PROGRAM PRG_SFLX_ValidationAsConfirmation
VAR
	rtrigValidCameraTrigger				: F_TRIG;
	bSideFlexValidCameraTrigger			: BOOL;

	rsSideFlexTwoOutersInAggregation	: RS;
	rsSideFlexPackToOuterProcessing		: RS;

	rtrigNewOuterArrived					: R_TRIG;
	bNewOuterIsProccesing				: BOOL;
	tonValidationTimout					: TON;
	bValidationTimeout					: BOOL;
	bValidationTimeoutReset				: BOOL;
	fbTimeoutCounter						: CTU;
	nCount									: WORD;


	fbOuterValidationCamera				: FB_SCANNER_CameraSelect;
	(*stOuterValidationCameraOptions		: ST_SCANNER_Options := (eScannerType := E_MV_420_FULL, nImageBuffer := 1, nExpectedResp := 2);*)
	fbOuterValidationEvaluation		: FB_SCANNER_Evaluation;

	fbCheckForDuplicateOuterValidation	: FB_OUTER_CheckDuplicateStatus;


	rtrigOuterValidationCameraDone				: R_TRIG;
	bOuterValidationCameraDone				: BOOL;
	bDataReadyForValidation			: BOOL;
	bQAReject							: BOOL;

	sLastImageLableString				: T_OUTER_Barcode;

	fbPerformance							: FB_Interval;
	fbMoveOuterData						: FB_OUTER_MoveOuterStatus;
	fbCompleteOuterFromQueue			: FB_OUTER_CompleteDataFromQueue_NoCam;
	fbMETSValidateOuterForReject			: FB_OUTER_ValidateOuterForReject;
	tofValidateOuterDoneForHMI			: TOF;
	fbMasterListUpdate					: FB_OUTER_MasterListUpdate;

	stLastOuterCompleted				: ST_OUTER_Status;
	sLastReadOuterBarcode			: T_OUTER_Barcode;
	nOutersCompleted					: UDINT;
	bDoneInfo							: BOOL;

	rtrigSetOuterValidationOK			: R_TRIG;
	rtrigSetOuterValidationNOK		: R_TRIG;

	rsOuterRejectStation 				: RS;
	rsOuterRejectConfirmation 		: RS;

	rtrigResetValidationStatus			: R_TRIG;

	sRejectCode						: STRING(255);
	fbArchiveInvalidOuters			: FB_OUTER_ArchiveInvalidOuters;
	aReasonForReject					: ARRAY[0..50] OF STRING(255);
	bClearList							: BOOL;

	fbOuterProduced					: FB_KPI_GenericEfficiency;
	fbOuterInspection					: FB_KPI_OutersEfficiency;

	stDummyImage					: ST_SCANNER_ImageData;

	fbOuterLevelCounter				: FB_KPI_OuterLevelCounter;

	fbQARejectCounter				: FB_CTU32;
	fbOuterValidationIndexOK			: FB_CTU32;

	ctuConsecutiveOuterRejects		: CTU;
	nActualCount						: WORD;
END_VAR
VAR // added by the converter: edge detectors and wires of the graphical bodies
    _w1 : E_CYLINDER_Position;
    _w2, _w3 : BOOL;
END_VAR

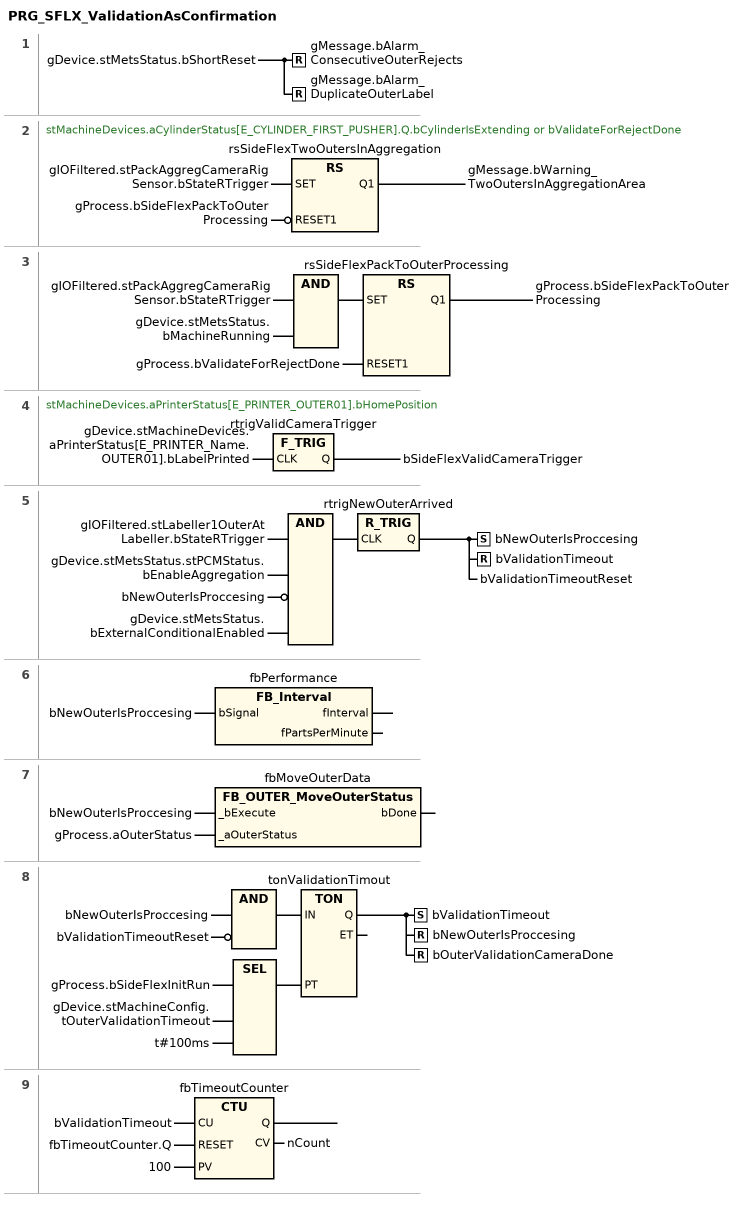
// NETWORK 1
gMessage.bAlarm_ConsecutiveOuterRejects R= gDevice.stMetsStatus.bShortReset;
gMessage.bAlarm_DuplicateOuterLabel R= gDevice.stMetsStatus.bShortReset;

// NETWORK 2
// stMachineDevices.aCylinderStatus[E_CYLINDER_FIRST_PUSHER].Q.bCylinderIsExtending or bValidateForRejectDone
rsSideFlexTwoOutersInAggregation(SET := gIOFiltered.stPackAggregCameraRigSensor.bStateRTrigger, RESET1 := NOT gProcess.bSideFlexPackToOuterProcessing); // RS
gMessage.bWarning_TwoOutersInAggregationArea := rsSideFlexTwoOutersInAggregation.Q1;

// NETWORK 3
rsSideFlexPackToOuterProcessing(SET := gIOFiltered.stPackAggregCameraRigSensor.bStateRTrigger AND gDevice.stMetsStatus.bMachineRunning, RESET1 := gProcess.bValidateForRejectDone); // RS
gProcess.bSideFlexPackToOuterProcessing := rsSideFlexPackToOuterProcessing.Q1;

// NETWORK 4
// stMachineDevices.aPrinterStatus[E_PRINTER_OUTER01].bHomePosition
rtrigValidCameraTrigger(CLK := gDevice.stMachineDevices.aPrinterStatus[E_PRINTER_Name.OUTER01].bLabelPrinted); // F_TRIG
bSideFlexValidCameraTrigger := rtrigValidCameraTrigger.Q;

// NETWORK 5
rtrigNewOuterArrived(CLK := gIOFiltered.stLabeller1OuterAtLabeller.bStateRTrigger AND gDevice.stMetsStatus.stPCMStatus.bEnableAggregation AND NOT bNewOuterIsProccesing AND gDevice.stMetsStatus.bExternalConditionalEnabled); // R_TRIG
bNewOuterIsProccesing S= rtrigNewOuterArrived.Q;
bValidationTimeout R= rtrigNewOuterArrived.Q;
bValidationTimeoutReset := rtrigNewOuterArrived.Q;

// NETWORK 6
fbPerformance(bSignal := bNewOuterIsProccesing); // FB_Interval

// NETWORK 7
fbMoveOuterData(_bExecute := bNewOuterIsProccesing, _aOuterStatus := gProcess.aOuterStatus); // FB_OUTER_MoveOuterStatus

// NETWORK 8
tonValidationTimout(IN := bNewOuterIsProccesing AND NOT bValidationTimeoutReset, PT := SEL(gProcess.bSideFlexInitRun, gDevice.stMachineConfig.tOuterValidationTimeout, t#100ms)); // TON
bValidationTimeout S= tonValidationTimout.Q;
bNewOuterIsProccesing R= tonValidationTimout.Q;
bOuterValidationCameraDone R= tonValidationTimout.Q;

// NETWORK 9
fbTimeoutCounter(CU := bValidationTimeout, RESET := fbTimeoutCounter.Q, PV := 100, CV => nCount); // CTU

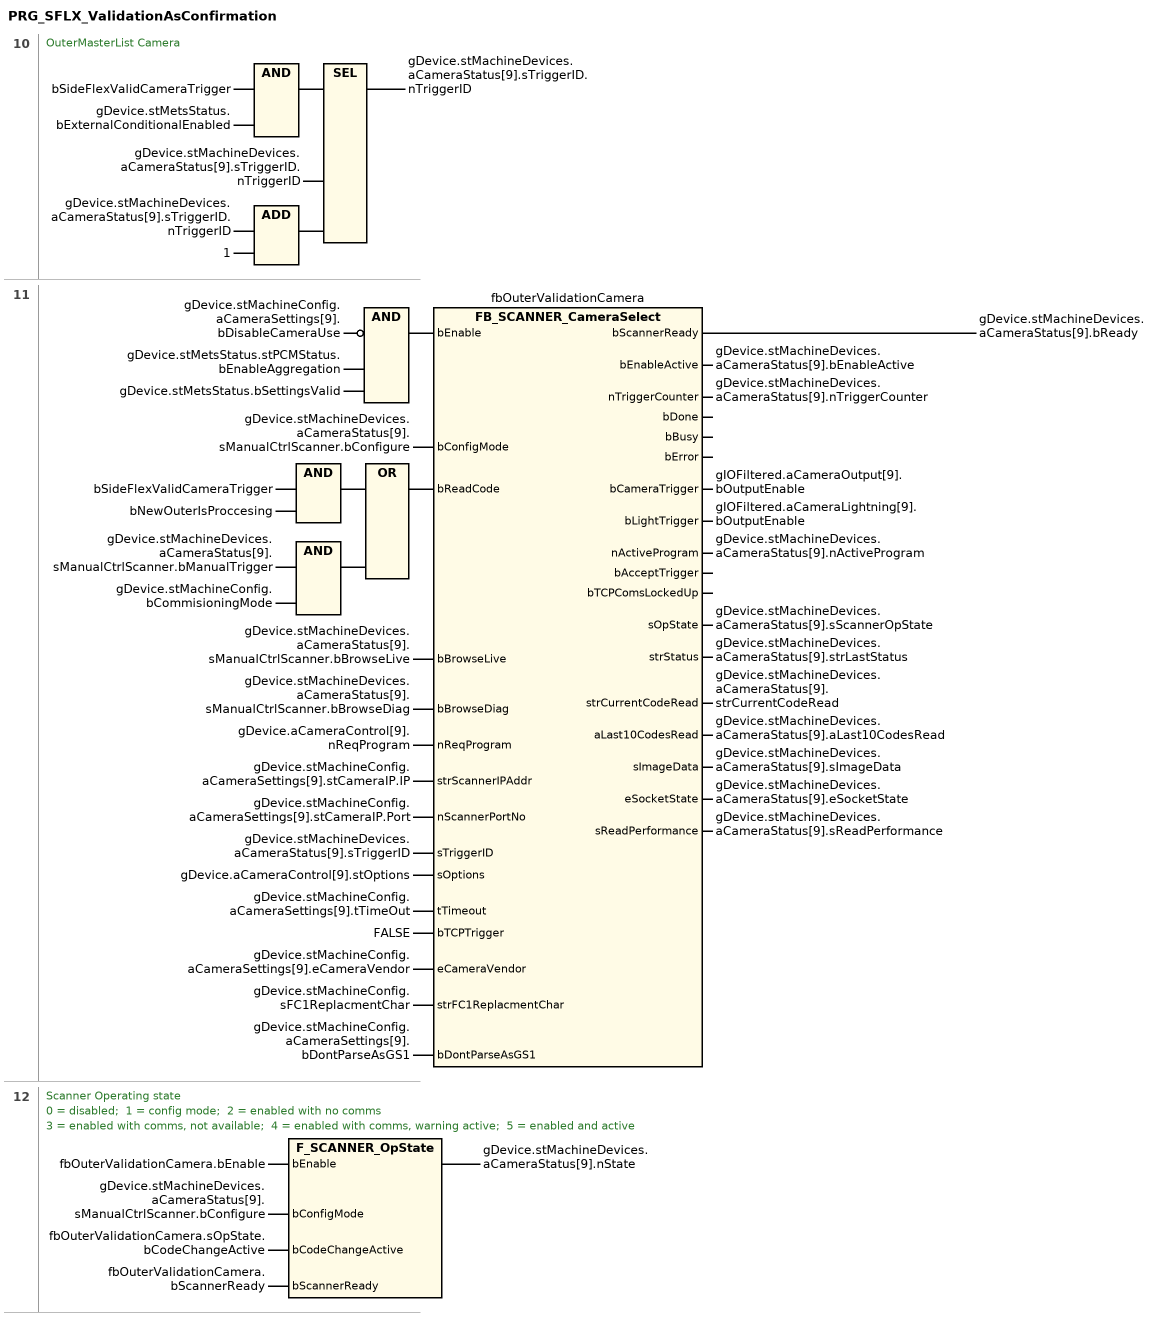
// NETWORK 10
// OuterMasterList Camera
gDevice.stMachineDevices.aCameraStatus[9].sTriggerID.nTriggerID := SEL(bSideFlexValidCameraTrigger AND gDevice.stMetsStatus.bExternalConditionalEnabled, gDevice.stMachineDevices.aCameraStatus[9].sTriggerID.nTriggerID, gDevice.stMachineDevices.aCameraStatus[9].sTriggerID.nTriggerID + 1);

// NETWORK 11
fbOuterValidationCamera(
    bEnable := NOT gDevice.stMachineConfig.aCameraSettings[9].bDisableCameraUse AND gDevice.stMetsStatus.stPCMStatus.bEnableAggregation AND gDevice.stMetsStatus.bSettingsValid,
    bConfigMode := gDevice.stMachineDevices.aCameraStatus[9].sManualCtrlScanner.bConfigure,
    bReadCode := bSideFlexValidCameraTrigger AND bNewOuterIsProccesing OR gDevice.stMachineDevices.aCameraStatus[9].sManualCtrlScanner.bManualTrigger AND gDevice.stMachineConfig.bCommisioningMode,
    bBrowseLive := gDevice.stMachineDevices.aCameraStatus[9].sManualCtrlScanner.bBrowseLive,
    bBrowseDiag := gDevice.stMachineDevices.aCameraStatus[9].sManualCtrlScanner.bBrowseDiag,
    nReqProgram := gDevice.aCameraControl[9].nReqProgram,
    strScannerIPAddr := gDevice.stMachineConfig.aCameraSettings[9].stCameraIP.IP,
    nScannerPortNo := gDevice.stMachineConfig.aCameraSettings[9].stCameraIP.Port,
    sTriggerID := gDevice.stMachineDevices.aCameraStatus[9].sTriggerID,
    sOptions := gDevice.aCameraControl[9].stOptions,
    tTimeout := gDevice.stMachineConfig.aCameraSettings[9].tTimeOut,
    bTCPTrigger := FALSE,
    eCameraVendor := gDevice.stMachineConfig.aCameraSettings[9].eCameraVendor,
    strFC1ReplacmentChar := gDevice.stMachineConfig.sFC1ReplacmentChar,
    bDontParseAsGS1 := gDevice.stMachineConfig.aCameraSettings[9].bDontParseAsGS1,
    bEnableActive => gDevice.stMachineDevices.aCameraStatus[9].bEnableActive,
    nTriggerCounter => gDevice.stMachineDevices.aCameraStatus[9].nTriggerCounter,
    bCameraTrigger => gIOFiltered.aCameraOutput[9].bOutputEnable,
    bLightTrigger => gIOFiltered.aCameraLightning[9].bOutputEnable,
    nActiveProgram => gDevice.stMachineDevices.aCameraStatus[9].nActiveProgram,
    sOpState => gDevice.stMachineDevices.aCameraStatus[9].sScannerOpState,
    strStatus => gDevice.stMachineDevices.aCameraStatus[9].strLastStatus,
    strCurrentCodeRead => gDevice.stMachineDevices.aCameraStatus[9].strCurrentCodeRead,
    aLast10CodesRead => gDevice.stMachineDevices.aCameraStatus[9].aLast10CodesRead,
    sImageData => gDevice.stMachineDevices.aCameraStatus[9].sImageData,
    eSocketState => gDevice.stMachineDevices.aCameraStatus[9].eSocketState,
    sReadPerformance => gDevice.stMachineDevices.aCameraStatus[9].sReadPerformance); // FB_SCANNER_CameraSelect
gDevice.stMachineDevices.aCameraStatus[9].bReady := fbOuterValidationCamera.bScannerReady;

// NETWORK 12
// 					Scanner Operating state
// 0 = disabled;  1 = config mode;  2 = enabled with no comms
// 3 = enabled with comms, not available;  4 = enabled with comms, warning active;  5 = enabled and active
//
gDevice.stMachineDevices.aCameraStatus[9].nState := F_SCANNER_OpState(bEnable := fbOuterValidationCamera.bEnable, bConfigMode := gDevice.stMachineDevices.aCameraStatus[9].sManualCtrlScanner.bConfigure, bCodeChangeActive := fbOuterValidationCamera.sOpState.bCodeChangeActive, bScannerReady := fbOuterValidationCamera.bScannerReady);

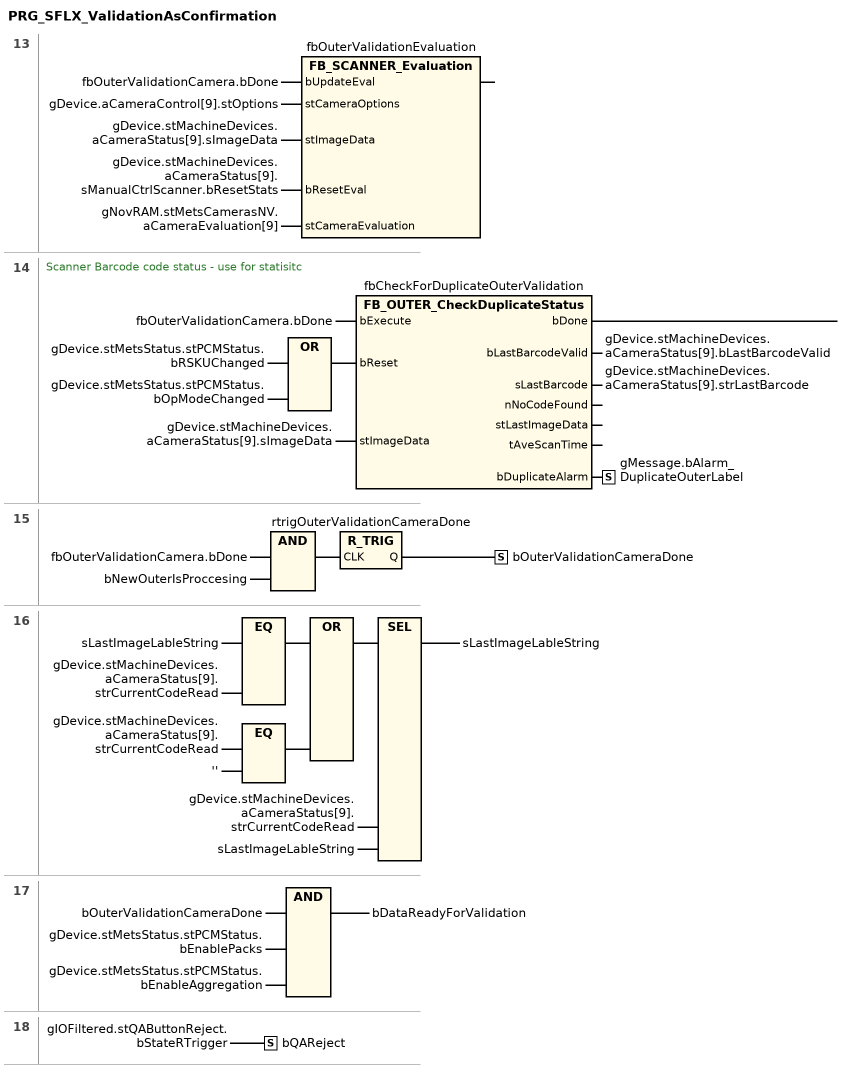
// NETWORK 13
fbOuterValidationEvaluation(
    bUpdateEval := fbOuterValidationCamera.bDone,
    stCameraOptions := gDevice.aCameraControl[9].stOptions,
    stImageData := gDevice.stMachineDevices.aCameraStatus[9].sImageData,
    bResetEval := gDevice.stMachineDevices.aCameraStatus[9].sManualCtrlScanner.bResetStats,
    stCameraEvaluation := gNovRAM.stMetsCamerasNV.aCameraEvaluation[9]); // FB_SCANNER_Evaluation

// NETWORK 14
// Scanner Barcode code status - use for statisitc
fbCheckForDuplicateOuterValidation(
    bExecute := fbOuterValidationCamera.bDone,
    bReset := gDevice.stMetsStatus.stPCMStatus.bRSKUChanged OR gDevice.stMetsStatus.stPCMStatus.bOpModeChanged,
    stImageData := gDevice.stMachineDevices.aCameraStatus[9].sImageData,
    bLastBarcodeValid => gDevice.stMachineDevices.aCameraStatus[9].bLastBarcodeValid,
    sLastBarcode => gDevice.stMachineDevices.aCameraStatus[9].strLastBarcode); // FB_OUTER_CheckDuplicateStatus
gMessage.bAlarm_DuplicateOuterLabel S= fbCheckForDuplicateOuterValidation.bDuplicateAlarm;

// NETWORK 15
rtrigOuterValidationCameraDone(CLK := fbOuterValidationCamera.bDone AND bNewOuterIsProccesing); // R_TRIG
bOuterValidationCameraDone S= rtrigOuterValidationCameraDone.Q;

// NETWORK 16
sLastImageLableString := SEL(sLastImageLableString = gDevice.stMachineDevices.aCameraStatus[9].strCurrentCodeRead OR gDevice.stMachineDevices.aCameraStatus[9].strCurrentCodeRead = '', gDevice.stMachineDevices.aCameraStatus[9].strCurrentCodeRead, sLastImageLableString);

// NETWORK 17
bDataReadyForValidation := bOuterValidationCameraDone AND gDevice.stMetsStatus.stPCMStatus.bEnablePacks AND gDevice.stMetsStatus.stPCMStatus.bEnableAggregation;

// NETWORK 18
bQAReject S= gIOFiltered.stQAButtonReject.bStateRTrigger;

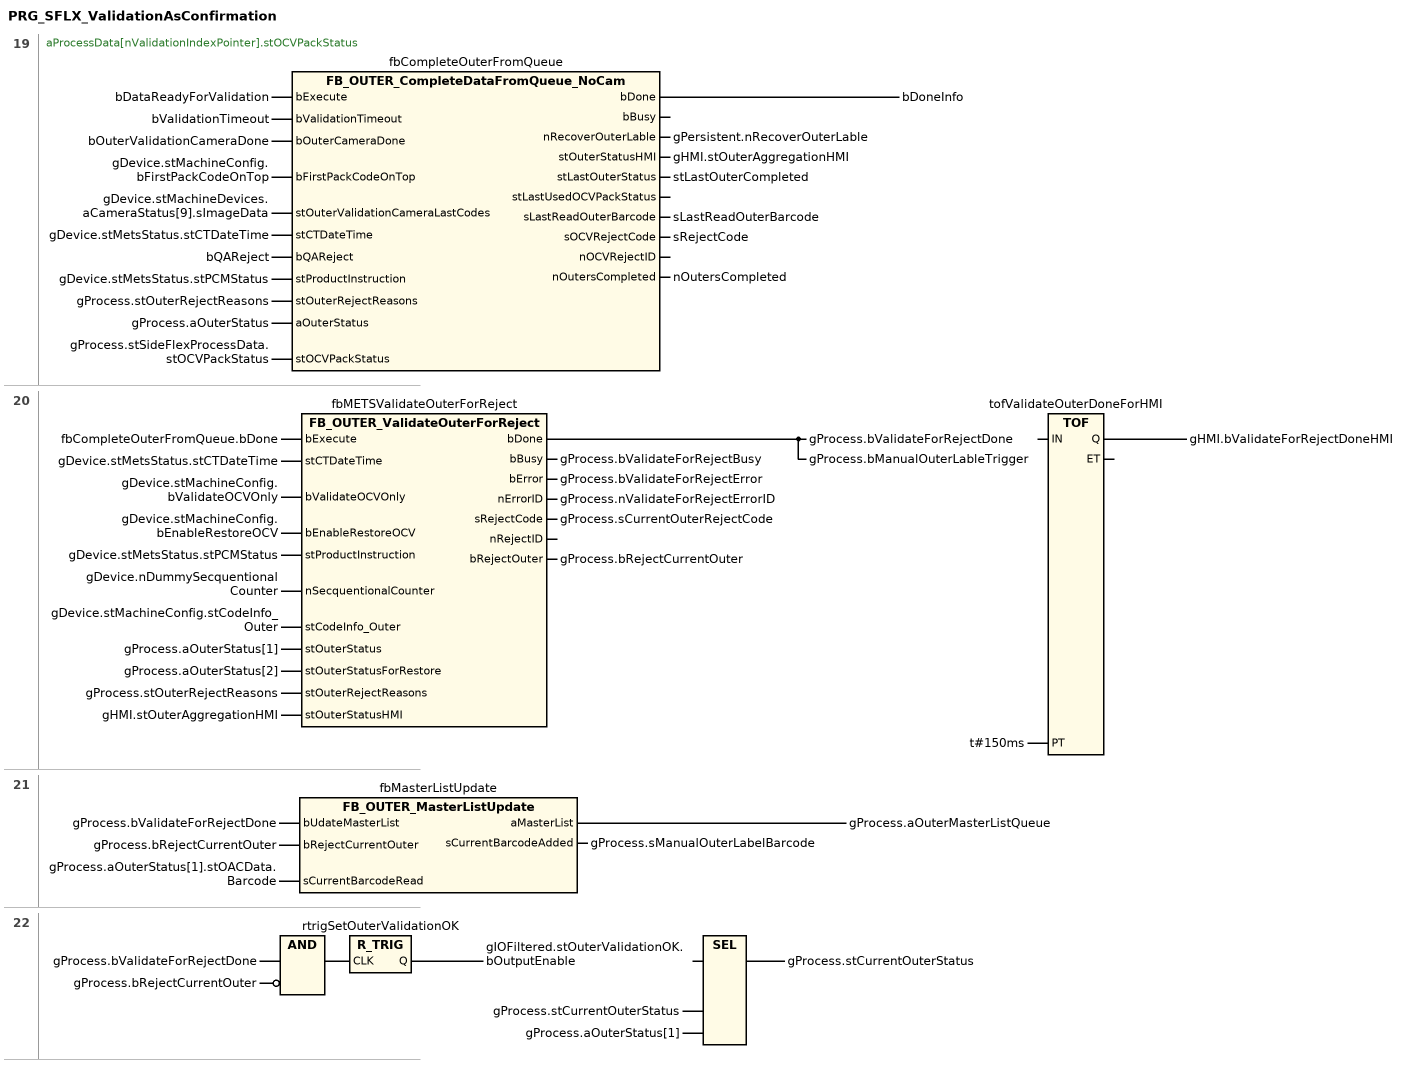
// NETWORK 19
// aProcessData[nValidationIndexPointer].stOCVPackStatus
fbCompleteOuterFromQueue(
    bExecute := bDataReadyForValidation,
    bValidationTimeout := bValidationTimeout,
    bOuterCameraDone := bOuterValidationCameraDone,
    bFirstPackCodeOnTop := gDevice.stMachineConfig.bFirstPackCodeOnTop,
    stOuterValidationCameraLastCodes := gDevice.stMachineDevices.aCameraStatus[9].sImageData,
    stCTDateTime := gDevice.stMetsStatus.stCTDateTime,
    bQAReject := bQAReject,
    stProductInstruction := gDevice.stMetsStatus.stPCMStatus,
    stOuterRejectReasons := gProcess.stOuterRejectReasons,
    aOuterStatus := gProcess.aOuterStatus,
    stOCVPackStatus := gProcess.stSideFlexProcessData.stOCVPackStatus,
    nRecoverOuterLable => gPersistent.nRecoverOuterLable,
    stOuterStatusHMI => gHMI.stOuterAggregationHMI,
    stLastOuterStatus => stLastOuterCompleted,
    sLastReadOuterBarcode => sLastReadOuterBarcode,
    sOCVRejectCode => sRejectCode,
    nOutersCompleted => nOutersCompleted); // FB_OUTER_CompleteDataFromQueue_NoCam
bDoneInfo := fbCompleteOuterFromQueue.bDone;

// NETWORK 20
fbMETSValidateOuterForReject(
    bExecute := fbCompleteOuterFromQueue.bDone,
    stCTDateTime := gDevice.stMetsStatus.stCTDateTime,
    bValidateOCVOnly := gDevice.stMachineConfig.bValidateOCVOnly,
    bEnableRestoreOCV := gDevice.stMachineConfig.bEnableRestoreOCV,
    stProductInstruction := gDevice.stMetsStatus.stPCMStatus,
    nSecquentionalCounter := gDevice.nDummySecquentionalCounter,
    stCodeInfo_Outer := gDevice.stMachineConfig.stCodeInfo_Outer,
    stOuterStatus := gProcess.aOuterStatus[1],
    stOuterStatusForRestore := gProcess.aOuterStatus[2],
    stOuterRejectReasons := gProcess.stOuterRejectReasons,
    stOuterStatusHMI := gHMI.stOuterAggregationHMI,
    bBusy => gProcess.bValidateForRejectBusy,
    bError => gProcess.bValidateForRejectError,
    nErrorID => gProcess.nValidateForRejectErrorID,
    sRejectCode => gProcess.sCurrentOuterRejectCode,
    bRejectOuter => gProcess.bRejectCurrentOuter); // FB_OUTER_ValidateOuterForReject
gProcess.bValidateForRejectDone := fbMETSValidateOuterForReject.bDone;
gProcess.bManualOuterLableTrigger := fbMETSValidateOuterForReject.bDone;
tofValidateOuterDoneForHMI(IN := fbMETSValidateOuterForReject.bDone, PT := t#150ms); // TOF
gHMI.bValidateForRejectDoneHMI := tofValidateOuterDoneForHMI.Q;

// NETWORK 21
fbMasterListUpdate(
    bUdateMasterList := gProcess.bValidateForRejectDone,
    bRejectCurrentOuter := gProcess.bRejectCurrentOuter,
    sCurrentBarcodeRead := gProcess.aOuterStatus[1].stOACData.Barcode,
    sCurrentBarcodeAdded => gProcess.sManualOuterLabelBarcode); // FB_OUTER_MasterListUpdate
gProcess.aOuterMasterListQueue := fbMasterListUpdate.aMasterList;

// NETWORK 22
rtrigSetOuterValidationOK(CLK := gProcess.bValidateForRejectDone AND NOT gProcess.bRejectCurrentOuter); // R_TRIG
gIOFiltered.stOuterValidationOK.bOutputEnable := rtrigSetOuterValidationOK.Q;
gProcess.stCurrentOuterStatus := SEL(rtrigSetOuterValidationOK.Q, gProcess.stCurrentOuterStatus, gProcess.aOuterStatus[1]);

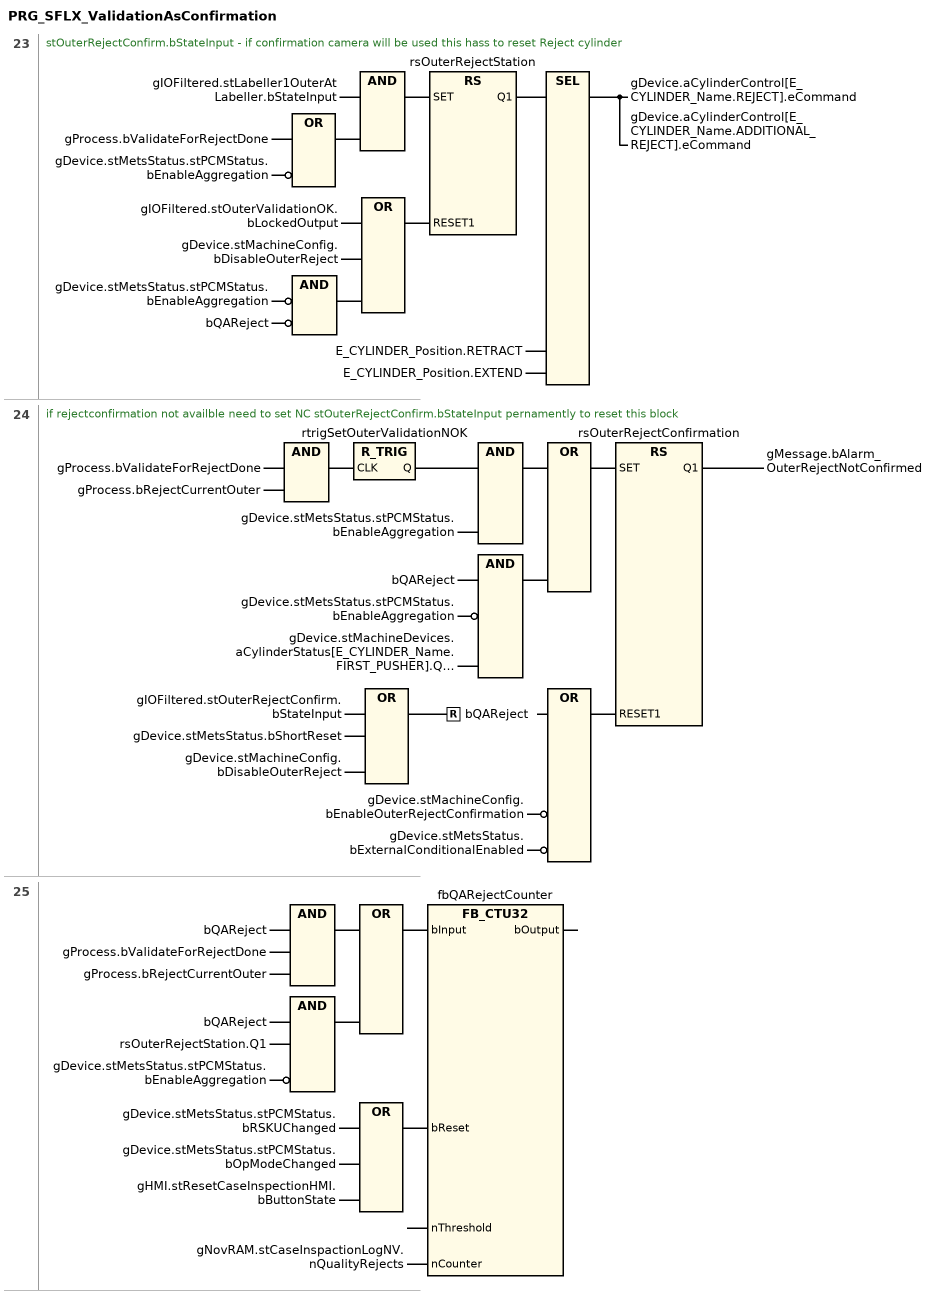
// NETWORK 23
// stOuterRejectConfirm.bStateInput - if confirmation camera will be used this hass to reset Reject cylinder
rsOuterRejectStation(SET := gIOFiltered.stLabeller1OuterAtLabeller.bStateInput AND (gProcess.bValidateForRejectDone OR NOT gDevice.stMetsStatus.stPCMStatus.bEnableAggregation), RESET1 := gIOFiltered.stOuterValidationOK.bLockedOutput OR gDevice.stMachineConfig.bDisableOuterReject OR NOT gDevice.stMetsStatus.stPCMStatus.bEnableAggregation AND NOT bQAReject); // RS
_w1 := SEL(rsOuterRejectStation.Q1, E_CYLINDER_Position.RETRACT, E_CYLINDER_Position.EXTEND);
gDevice.aCylinderControl[E_CYLINDER_Name.REJECT].eCommand := _w1;
gDevice.aCylinderControl[E_CYLINDER_Name.ADDITIONAL_REJECT].eCommand := _w1;

// NETWORK 24
// if rejectconfirmation not availble need to set NC stOuterRejectConfirm.bStateInput pernamently to reset this block
rtrigSetOuterValidationNOK(CLK := gProcess.bValidateForRejectDone AND gProcess.bRejectCurrentOuter); // R_TRIG
_w3 := rtrigSetOuterValidationNOK.Q AND gDevice.stMetsStatus.stPCMStatus.bEnableAggregation OR bQAReject AND NOT gDevice.stMetsStatus.stPCMStatus.bEnableAggregation AND gDevice.stMachineDevices.aCylinderStatus[E_CYLINDER_Name.FIRST_PUSHER].Q.bCylinderInExtendedPosition;
_w2 := gIOFiltered.stOuterRejectConfirm.bStateInput OR gDevice.stMetsStatus.bShortReset OR gDevice.stMachineConfig.bDisableOuterReject;
bQAReject R= _w2;
rsOuterRejectConfirmation(SET := _w3, RESET1 := _w2 OR NOT gDevice.stMachineConfig.bEnableOuterRejectConfirmation OR NOT gDevice.stMetsStatus.bExternalConditionalEnabled); // RS
gMessage.bAlarm_OuterRejectNotConfirmed := rsOuterRejectConfirmation.Q1;

// NETWORK 25
fbQARejectCounter(
    bInput := bQAReject AND gProcess.bValidateForRejectDone AND gProcess.bRejectCurrentOuter OR bQAReject AND rsOuterRejectStation.Q1 AND NOT gDevice.stMetsStatus.stPCMStatus.bEnableAggregation,
    bReset := gDevice.stMetsStatus.stPCMStatus.bRSKUChanged OR gDevice.stMetsStatus.stPCMStatus.bOpModeChanged OR gHMI.stResetCaseInspectionHMI.bButtonState,
    nCounter := gNovRAM.stCaseInspactionLogNV.nQualityRejects); // FB_CTU32

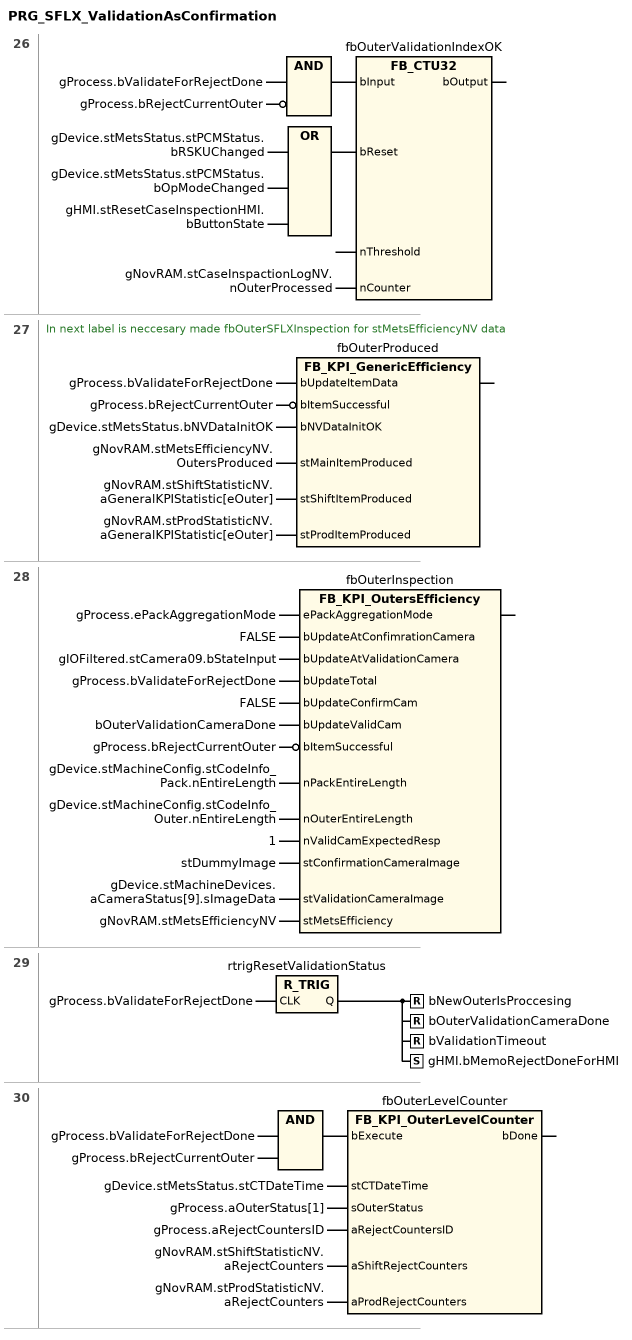
// NETWORK 26
fbOuterValidationIndexOK(
    bInput := gProcess.bValidateForRejectDone AND NOT gProcess.bRejectCurrentOuter,
    bReset := gDevice.stMetsStatus.stPCMStatus.bRSKUChanged OR gDevice.stMetsStatus.stPCMStatus.bOpModeChanged OR gHMI.stResetCaseInspectionHMI.bButtonState,
    nCounter := gNovRAM.stCaseInspactionLogNV.nOuterProcessed); // FB_CTU32

// NETWORK 27
// In next label is neccesary made fbOuterSFLXInspection for stMetsEfficiencyNV data
fbOuterProduced(
    bUpdateItemData := gProcess.bValidateForRejectDone,
    bItemSuccessful := NOT gProcess.bRejectCurrentOuter,
    bNVDataInitOK := gDevice.stMetsStatus.bNVDataInitOK,
    stMainItemProduced := gNovRAM.stMetsEfficiencyNV.OutersProduced,
    stShiftItemProduced := gNovRAM.stShiftStatisticNV.aGeneralKPIStatistic[eOuter],
    stProdItemProduced := gNovRAM.stProdStatisticNV.aGeneralKPIStatistic[eOuter]); // FB_KPI_GenericEfficiency

// NETWORK 28
fbOuterInspection(
    ePackAggregationMode := gProcess.ePackAggregationMode,
    bUpdateAtConfimrationCamera := FALSE,
    bUpdateAtValidationCamera := gIOFiltered.stCamera09.bStateInput,
    bUpdateTotal := gProcess.bValidateForRejectDone,
    bUpdateConfirmCam := FALSE,
    bUpdateValidCam := bOuterValidationCameraDone,
    bItemSuccessful := NOT gProcess.bRejectCurrentOuter,
    nPackEntireLength := gDevice.stMachineConfig.stCodeInfo_Pack.nEntireLength,
    nOuterEntireLength := gDevice.stMachineConfig.stCodeInfo_Outer.nEntireLength,
    nValidCamExpectedResp := 1,
    stConfirmationCameraImage := stDummyImage,
    stValidationCameraImage := gDevice.stMachineDevices.aCameraStatus[9].sImageData,
    stMetsEfficiency := gNovRAM.stMetsEfficiencyNV); // FB_KPI_OutersEfficiency

// NETWORK 29
rtrigResetValidationStatus(CLK := gProcess.bValidateForRejectDone); // R_TRIG
bNewOuterIsProccesing R= rtrigResetValidationStatus.Q;
bOuterValidationCameraDone R= rtrigResetValidationStatus.Q;
bValidationTimeout R= rtrigResetValidationStatus.Q;
gHMI.bMemoRejectDoneForHMI S= rtrigResetValidationStatus.Q;

// NETWORK 30
fbOuterLevelCounter(
    bExecute := gProcess.bValidateForRejectDone AND gProcess.bRejectCurrentOuter,
    stCTDateTime := gDevice.stMetsStatus.stCTDateTime,
    sOuterStatus := gProcess.aOuterStatus[1],
    aRejectCountersID := gProcess.aRejectCountersID,
    aShiftRejectCounters := gNovRAM.stShiftStatisticNV.aRejectCounters,
    aProdRejectCounters := gNovRAM.stProdStatisticNV.aRejectCounters); // FB_KPI_OuterLevelCounter

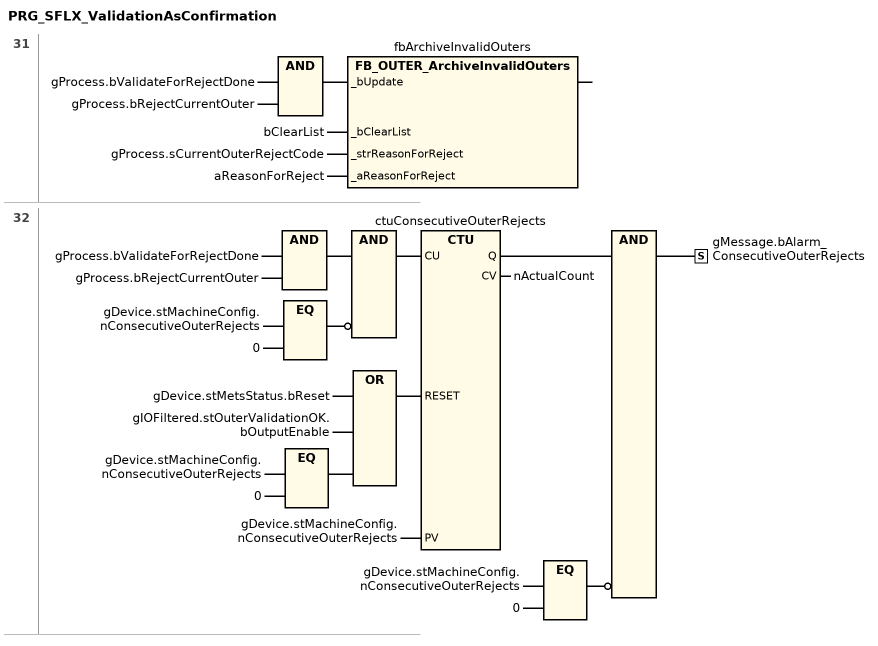
// NETWORK 31
fbArchiveInvalidOuters(
    _bUpdate := gProcess.bValidateForRejectDone AND gProcess.bRejectCurrentOuter,
    _bClearList := bClearList,
    _strReasonForReject := gProcess.sCurrentOuterRejectCode,
    _aReasonForReject := aReasonForReject); // FB_OUTER_ArchiveInvalidOuters

// NETWORK 32
ctuConsecutiveOuterRejects(
    CU := (gProcess.bValidateForRejectDone AND gProcess.bRejectCurrentOuter) AND NOT (gDevice.stMachineConfig.nConsecutiveOuterRejects = 0),
    RESET := gDevice.stMetsStatus.bReset OR gIOFiltered.stOuterValidationOK.bOutputEnable OR gDevice.stMachineConfig.nConsecutiveOuterRejects = 0,
    PV := gDevice.stMachineConfig.nConsecutiveOuterRejects,
    CV => nActualCount); // CTU
gMessage.bAlarm_ConsecutiveOuterRejects S= ctuConsecutiveOuterRejects.Q AND NOT (gDevice.stMachineConfig.nConsecutiveOuterRejects = 0);

END_PROGRAM

(* stored: Version 1.1.0.1
   POU PRG_SFLX_ValidationAsConfirmation: Id {0ecbf956-eefe-47d0-8936-ad1ff1b90aab}, SpecialFunc None *)
